{attribute 'call_after_init'}
FUNCTION_BLOCK FINAL TimeParam EXTENDS BaseParam
VAR_INPUT
END_VAR
VAR_OUTPUT
	value: TIME;
END_VAR
VAR
END_VAR

METHOD Change_Param
VAR_INPUT
	value	: STRING;
END_VAR
VAR
	_last_char: STRING;
	_value_ms: DWORD;
END_VAR
//This method changes the TIME value. It accepts more TIME formats than standard T#12s.
//Accepted formats include:
// - 12s, 12S, 12 s, 12 S, T#12S, T#12s, T#0m12S, 12000, etc

value := F_ToLCase(value);

WHILE FIND(value, ' ') <> 0 DO
	value := DELETE(value, 1, FIND(value, ' '));
END_WHILE

_last_char := RIGHT(value, 1);
IF _last_char <> 's' AND _last_char <> 'm' AND _last_char <> 'h' AND _last_char <> 'd' THEN
	_value_ms := STRING_TO_DWORD(value);
	value := DWORD_TO_STRING(_value_ms);
	value := concat(value, 'ms');
END_IF

value := DELETE(value, 1, FIND(value, 't#'));
value := CONCAT('T#', value);

THIS^.value := STRING_TO_TIME(value);
_display := TIME_TO_STRING(THIS^.value);
_display := DELETE(_display, 2, 1);
END_METHOD

METHOD Quick_Change
VAR_INPUT
	value: TIME;
END_VAR
THIS^.value := value;
_display := TIME_TO_STRING(THIS^.value);
_display := DELETE(_display, 2, 1);
END_METHOD

END_FUNCTION_BLOCK

(* stored: Version 1.1.0.1, ProductVersion 3.1.4024.12
   POU TimeParam: Id {e42b2b62-7024-4947-950d-1bbb2145cbdf}, SpecialFunc None
   Method Change_Param: Id {b8a78d61-360c-4d46-83bb-bf1dc6cf7dbe}
   Method Quick_Change: Id {4e207cf7-d870-4cd3-86ab-7e71fa397efc} *)
